PROGRAM VltLadder_Shapes
VAR
	a : BOOL;
	b : BOOL;
	c : BOOL;
	out1 : BOOL;
	out2 : BOOL;
END_VAR

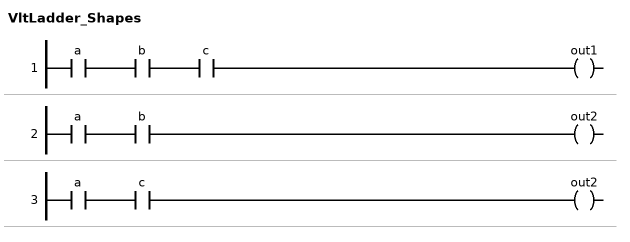
// NETWORK 1
out1 := (a AND b) AND c;

// NETWORK 2
out2 := a AND b;

// NETWORK 3
out2 := a AND c;

END_PROGRAM

(* stored: Version 1.1.0.1, ProductVersion 3.1.4024.16
   POU VltLadder_Shapes: Id {af09489d-96d3-4c46-b21e-e0cc39b26cd8}, SpecialFunc None *)
